// TIA Portal V17 export
// export: Created 2025-08-05T09:36:01.1535554Z, ExportSetting WithDefaults, DisplayName Totally Integrated Automation Portal, DisplayVersion V17, DisplayName TIA Portal Openness, DisplayVersion V17, DisplayName TIA Portal Version Control Interface, DisplayVersion V17, DisplayName SINAMICS Startdrive Advanced, DisplayVersion V17, DisplayName SINAMICS Startdrive G130, G150, S120, S150, SINAMICS MV, S210, DisplayVersion V17, DisplayName SINAMICS Startdrive G110M, G120, G120C, G120D, G120P, G115D, DisplayVersion V17, DisplayName STEP 7 Professional, DisplayVersion V17, DisplayName STEP 7 Safety, DisplayVersion V17, DisplayName WinCC Advanced, DisplayVersion V17
TYPE "typeMotionOvrvList"
TITLE = Motion overview list / Motion-Übersichtsliste
// Motion overview list [V 01.00 | Kernel_V2] / Motion-Übersichtsliste [V 01.00 | Kernel_V2]
// stored: IsFailsafeCompliant false
   STRUCT
      enabled : Bool;   // Motion-Übersicht ist freigeschaltet / Motion overview is activated
      lastUsedIndex : DInt := -1;   // Letzter Benutzter Index / Last user index
      valid : Bool;   // Gültigkeit / Scope
      overflowCount : DInt;   // Gruppen Überlauf Zähler / Groups overtravel counter
      motions : Array[0.."MAX_CNT_MTN_OVR_ENTRIES"] of "typeMotionOvrvListEntry";   // Motions
   END_STRUCT;
END_TYPE
